FUNCTION RadiansToDegrees : LREAL
VAR_INPUT
	radians : LREAL;
END_VAR
VAR
END_VAR

RadiansToDegrees := radians * 180 / GVL_RobotArmConstants.Pi;

END_FUNCTION

(* stored: Version 1.1.0.1, ProductVersion 3.1.4024.12
   POU RadiansToDegrees: Id {3bc61a45-1381-43a2-901e-4e4aca3a91d0}, SpecialFunc None *)
